// Library/Structures/Cartesian/RobotCartesianPosition
{attribute 'pack_mode' := '1'} 
// ------------------------------------------------------------------------- 
//  SRCI Robot Library                                                
// ------------------------------------------------------------------------- 
//                                                                           
//  Object:      RobotCartesianPosition                                       
//  Author:      Thorsten Brach                                                
//  Date:        2024-06-01
//
//  Description:                                              
//   
//                                                                           
//  Copyright: 
//    (C) 2024 Thorsten Brach. All rights reserved                                                                                                                                            
//             Licensed under the LGPL-3.0 license.
//                                                                           
//  Disclaimer:                                                                           
//    This project is provided without any guarantee and can be used for   
//    private and commercial purposes. Any use is at the user’s 
//    own risk and responsibility.
//
// -------------------------------------------------------------------------
TYPE RobotCartesianPosition EXTENDS RobotCartesianPositionShort : 
STRUCT
  /// Position of second external axis
  E2         : REAL;
  /// Position of third external axis
  E3         : REAL;
  /// Position of fourth external axis
  E4         : REAL;
  /// Position of fifth external axis
  E5         : REAL;
  /// Position of sixth external axis
  E6         : REAL;    
END_STRUCT
END_TYPE

// Library/Structures/Cartesian/RobotCartesianPositionBase
{attribute 'pack_mode' := '1'} 
// ------------------------------------------------------------------------- 
//  SRCI Robot Library                                                
// ------------------------------------------------------------------------- 
//                                                                           
//  Object:      RobotCartesianPosition                                       
//  Author:      Thorsten Brach                                                
//  Date:        2024-06-01
//
//  Description:                                              
//   
//                                                                           
//  Copyright: 
//    (C) 2024 Thorsten Brach. All rights reserved                                                                                                                                            
//             Licensed under the LGPL-3.0 license.
//                                                                           
//  Disclaimer:                                                                           
//    This project is provided without any guarantee and can be used for   
//    private and commercial purposes. Any use is at the user’s 
//    own risk and responsibility.
//
// -------------------------------------------------------------------------
TYPE RobotCartesianPositionBase :
STRUCT
  /// TCP Position on the X-Axis
  X          : REAL;
  /// TCP Position on the Y-Axis
  Y          : REAL;
  /// TCP Position on the Z-Axis
  Z          : REAL;
  /// Rotation around the X-Axis (RX)
  Rx         : REAL;
  /// Rotation around the Y-Axis (RY)
  Ry         : REAL;
  /// Rotation around the Z-Axis (RZ)
  Rz         : REAL;
END_STRUCT
END_TYPE

// Library/Structures/Cartesian/RobotCartesianPositionExt
{attribute 'pack_mode' := '1'} 
// ------------------------------------------------------------------------- 
//  SRCI Robot Library                                                
// ------------------------------------------------------------------------- 
//                                                                           
//  Object:      RobotCartesianPositionExt                                       
//  Author:      Thorsten Brach                                                
//  Date:        2024-06-01
//
//  Description:                                              
//   
//                                                                           
//  Copyright: 
//    (C) 2024 Thorsten Brach. All rights reserved                                                                                                                                            
//             Licensed under the LGPL-3.0 license.
//                                                                           
//  Disclaimer:                                                                           
//    This project is provided without any guarantee and can be used for   
//    private and commercial purposes. Any use is at the user’s 
//    own risk and responsibility.
//
// -------------------------------------------------------------------------
TYPE RobotCartesianPositionExt :
STRUCT
  /// Position of second external axis
  E2 : REAL;
  /// Position of third external axis
  E3 : REAL;
  /// Position of fourth external axis
  E4 : REAL;
  /// Position of fifth external axis
  E5 : REAL;
  /// Position of sixth external axis
  E6 : REAL;  
END_STRUCT
END_TYPE

// Library/Structures/Cartesian/RobotCartesianPositionShort
{attribute 'pack_mode' := '1'} 
// ------------------------------------------------------------------------- 
//  SRCI Robot Library                                                
// ------------------------------------------------------------------------- 
//                                                                           
//  Object:      RobotCartesianPositionShort                                       
//  Author:      Thorsten Brach                                                
//  Date:        2024-06-01
//
//  Description:                                              
//   
//                                                                           
//  Copyright: 
//    (C) 2024 Thorsten Brach. All rights reserved                                                                                                                                            
//             Licensed under the LGPL-3.0 license.
//                                                                           
//  Disclaimer:                                                                           
//    This project is provided without any guarantee and can be used for   
//    private and commercial purposes. Any use is at the user’s 
//    own risk and responsibility.
//
// -------------------------------------------------------------------------
TYPE RobotCartesianPositionShort EXTENDS RobotCartesianPositionBase:
STRUCT
  /// Configuration data of the robot (Config)
  Config     : ArmConfigParameter;
  /// Turn number of the axes (TurnNumber)
  TurnNumber : TurnNumber;
  /// Position of first external axis
  E1         : REAL;
END_STRUCT
END_TYPE

// Library/Structures/Common/CmdHeader
{attribute 'pack_mode' := '1'}
// ------------------------------------------------------------------------- 
//  SRCI Robot Library                                                
// ------------------------------------------------------------------------- 
//                                                                           
//  Object:      CmdHeader                                       
//  Author:      Thorsten Brach                                                
//  Date:        2024-06-01
//
//  Description:                                              
//   
//                                                                           
//  Copyright: 
//    (C) 2024 Thorsten Brach. All rights reserved                                                                                                                                            
//             Licensed under the LGPL-3.0 license.
//                                                                           
//  Disclaimer:                                                                           
//    This project is provided without any guarantee and can be used for   
//    private and commercial purposes. Any use is at the user’s 
//    own risk and responsibility.
//
// ------------------------------------------------------------------------- 
TYPE CmdHeader :
STRUCT
  /// Type of command - For more information see chapter 5.6.4.
 CmdTyp          : CmdType;
 /// Specifies target buffer and processing behavior - For more information see chapter 5.6.4.5
 ExecMode        : ExecutionMode;
 /// Parameter Sequence, used to identify sets of CMD parameter
 ParSeq          : BYTE;
 /// Priority of this command
 Priority        : PriorityLevel;  
END_STRUCT
END_TYPE

// Library/Structures/Common/LogParameter
{attribute 'pack_mode' := '1'} 
// ------------------------------------------------------------------------- 
//  SRCI Robot Library                                                
// ------------------------------------------------------------------------- 
//                                                                           
//  Object:      LogParameter                                       
//  Author:      Thorsten Brach                                                
//  Date:        2024-06-01
//
//  Description:                                              
//   
//                                                                           
//  Copyright: 
//    (C) 2024 Thorsten Brach. All rights reserved                                                                                                                                            
//             Licensed under the LGPL-3.0 license.
//                                                                           
//  Disclaimer:                                                                           
//    This project is provided without any guarantee and can be used for   
//    private and commercial purposes. Any use is at the user’s 
//    own risk and responsibility.
//
// -------------------------------------------------------------------------
TYPE LogParameter :
STRUCT
  /// Log level setting for creating commands  
  CreateCmd : LogLevel;
  /// Log level setting for updating commands
  UpdateCmd : LogLevel;
  /// Log level setting for generating sequence 
  GenSeq    : LogLevel;
  /// Log level for ??? sequence
  DecSeq    : LogLevel;
END_STRUCT
END_TYPE

// Library/Structures/Common/RobotCoordinateSystemParameters
{attribute 'pack_mode' := '1'} 
// ------------------------------------------------------------------------- 
//  SRCI Robot Library                                                
// ------------------------------------------------------------------------- 
//                                                                           
//  Object:      RobotCoordinateSystemParameters                                       
//  Author:      Thorsten Brach                                                
//  Date:        2024-06-01
//
//  Description:                                              
//   
//                                                                           
//  Copyright: 
//    (C) 2024 Thorsten Brach. All rights reserved                                                                                                                                            
//             Licensed under the LGPL-3.0 license.
//                                                                           
//  Disclaimer:                                                                           
//    This project is provided without any guarantee and can be used for   
//    private and commercial purposes. Any use is at the user’s 
//    own risk and responsibility.
//
// -------------------------------------------------------------------------
TYPE RobotCoordinateSystemParameters :
STRUCT
  /// Index of target tool
  /// • 0: Flange (default)
  /// • 1..254: Tool frames
  ToolNo : USINT;
  /// Index of target frame
  /// • 0: WCS (default)
  /// • 1..254: User frames
  FrameNo : USINT;  
END_STRUCT
END_TYPE

// Library/Structures/Common/RspHeader
{attribute 'pack_mode' := '1'}
// ------------------------------------------------------------------------- 
//  SRCI Robot Library                                                
// ------------------------------------------------------------------------- 
//                                                                           
//  Object:      RspHeader                                       
//  Author:      Thorsten Brach                                                
//  Date:        2024-06-01
//
//  Description:                                              
//   
//                                                                           
//  Copyright: 
//    (C) 2024 Thorsten Brach. All rights reserved                                                                                                                                            
//             Licensed under the LGPL-3.0 license.
//                                                                           
//  Disclaimer:                                                                           
//    This project is provided without any guarantee and can be used for   
//    private and commercial purposes. Any use is at the user’s 
//    own risk and responsibility.
//
// -------------------------------------------------------------------------
TYPE RspHeader :  
STRUCT
  /// Parameter Sequence, used to identify sets of CMD parameter - For more information see chapter 5.6.4
  ParSeq               : USINT;
  /// Actual state of the command - For more information and examples, see chapter 5.6.3.2
  State                : CmdMessageState;
  /// Severity of returned message according to .Table 5-47.
  AlarmMessageSeverity : Severity;
  /// Message code for error/warning/info identification reported during execution of command according to
  /// • Error: Table 7-1
  /// • Warning: Table 7-3
  /// • Info: Table 7-5
  AlarmMessageCode     : UINT;  
END_STRUCT
END_TYPE

// Library/Structures/Common/TimeStamp
{attribute 'pack_mode' := '1'} 
// ------------------------------------------------------------------------- 
//  SRCI Robot Library                                                
// ------------------------------------------------------------------------- 
//                                                                           
//  Object:      TimeStamp                                       
//  Author:      Thorsten Brach                                                
//  Date:        2024-06-01
//
//  Description:                                              
//   
//                                                                           
//  Copyright: 
//    (C) 2024 Thorsten Brach. All rights reserved                                                                                                                                            
//             Licensed under the LGPL-3.0 license.
//                                                                           
//  Disclaimer:                                                                           
//    This project is provided without any guarantee and can be used for   
//    private and commercial purposes. Any use is at the user’s 
//    own risk and responsibility.
//
// -------------------------------------------------------------------------
TYPE TimeStamp :
STRUCT
  /// Date of the timestamp
  TsData : IEC_DATE;
  /// Time of the timestamp
  TsTime : IEC_TIME;
END_STRUCT
END_TYPE

// Library/Structures/Data/CyclicStateData
{attribute 'pack_mode' := '1'} 
// ------------------------------------------------------------------------- 
//  SRCI Robot Library                                                
// ------------------------------------------------------------------------- 
//                                                                           
//  Object:      CyclicStateData                                       
//  Author:      Thorsten Brach                                                
//  Date:        2024-06-01
//
//  Description:                                              
//   
//                                                                           
//  Copyright: 
//    (C) 2024 Thorsten Brach. All rights reserved                                                                                                                                            
//             Licensed under the LGPL-3.0 license.
//                                                                           
//  Disclaimer:                                                                           
//    This project is provided without any guarantee and can be used for   
//    private and commercial purposes. Any use is at the user’s 
//    own risk and responsibility.
//
// -------------------------------------------------------------------------
TYPE CyclicStateData :
STRUCT
  /// Combination of various RA related states.
  StatusWord : RaStatusWord;
  /// Actual override in percentage multiplied by 100 (see chapter 5.6.2 for more information about the percentage encoding)
  Override   : UINT;
END_STRUCT
END_TYPE

// Library/Structures/Data/FrameData
{attribute 'pack_mode' := '1'} 
// ------------------------------------------------------------------------- 
//  SRCI Robot Library                                                
// ------------------------------------------------------------------------- 
//                                                                           
//  Object:      FrameData                                       
//  Author:      Thorsten Brach                                                
//  Date:        2024-06-01
//
//  Description:                                              
//   
//                                                                           
//  Copyright: 
//    (C) 2024 Thorsten Brach. All rights reserved                                                                                                                                            
//             Licensed under the LGPL-3.0 license.
//                                                                           
//  Disclaimer:                                                                           
//    This project is provided without any guarantee and can be used for   
//    private and commercial purposes. Any use is at the user’s 
//    own risk and responsibility.
//
// -------------------------------------------------------------------------
TYPE FrameData :
STRUCT
  /// Timestamp
  Timestamp      : IEC_TIMESTAMP;
  /// Frame to which the shifting and rotation is relative M
  ReferenceFrame : USINT;
  /// Origin of the coordinate system relative to the BCS/WCS/UCS 
  /// X value [mm]  
  X              : REAL := 0;
  /// Origin of the coordinate system relative to the BCS/WCS/UCS 
  /// Y value [mm]  
  Y              : REAL := 0;
  /// Origin of the coordinate system relative to the BCS/WCS/UCS 
  /// Z value [mm]  
  Z              : REAL := 0;
  /// Orientation of the coordinate system relative to the BCS/WCS/UCS
  /// Rx value [°]  
  Rx             : REAL := 0;
  /// Rx value [°]  
  Ry             : REAL := 0;
  /// Rx value [°]  
  Rz             : REAL := 0;  
END_STRUCT
END_TYPE

// Library/Structures/Data/LoadData
{attribute 'pack_mode' := '1'} 
// ------------------------------------------------------------------------- 
//  SRCI Robot Library                                                
// ------------------------------------------------------------------------- 
//                                                                           
//  Object:      LoadData                                       
//  Author:      Thorsten Brach                                                
//  Date:        2024-06-01
//
//  Description:                                              
//   
//                                                                           
//  Copyright: 
//    (C) 2024 Thorsten Brach. All rights reserved                                                                                                                                            
//             Licensed under the LGPL-3.0 license.
//                                                                           
//  Disclaimer:                                                                           
//    This project is provided without any guarantee and can be used for   
//    private and commercial purposes. Any use is at the user’s 
//    own risk and responsibility.
//
// -------------------------------------------------------------------------
TYPE LoadData :
STRUCT
  /// Timestamp
  Timestamp : IEC_TIMESTAMP;
  /// Position of the center of gravity relative to the flange.
  /// X value [mm]  
  X         : REAL := 0;
  /// Position of the center of gravity relative to the flange.
  /// Y value [mm]  
  Y         : REAL := 0;
  /// Position of the center of gravity relative to the flange.
  /// Z value [mm]  
  Z         : REAL := 0;
  /// Orientation of the principal inertia axes relative to the flange. O
  /// Rx value [°]  
  Rx        : REAL := 0;
  /// Ry value [°]  
  Ry        : REAL := 0;
  /// Rz value [°]  
  Rz        : REAL := 0;
  /// The mass of the tool and workpiece being gripped. [kg]
  Mass      : REAL := 0;
  /// The moment of inertia of the load around the resulting inertia X-Axis [kg/m²]
  Ix        : REAL := 0;
  /// The moment of inertia of the load around the resulting inertia y-axis [kg/m²]
  Iy        : REAL := 0;
  /// The moment of inertia of the load around the resulting inertia z-axis [kg/m²]
  Iz        : REAL := 0;  
END_STRUCT
END_TYPE

// Library/Structures/Data/RobotSubProgramData
{attribute 'pack_mode' := '1'} 
// ------------------------------------------------------------------------- 
//  SRCI Robot Library                                                
// ------------------------------------------------------------------------- 
//                                                                           
//  Object:      RobotSubProgramData                                       
//  Author:      Thorsten Brach                                                
//  Date:        2024-06-01
//
//  Description:                                              
//   
//                                                                           
//  Copyright: 
//    (C) 2024 Thorsten Brach. All rights reserved                                                                                                                                            
//             Licensed under the LGPL-3.0 license.
//                                                                           
//  Disclaimer:                                                                           
//    This project is provided without any guarantee and can be used for   
//    private and commercial purposes. Any use is at the user’s 
//    own risk and responsibility.
//
// -------------------------------------------------------------------------
TYPE RobotSubProgramData :
STRUCT
  /// Sub program data
  Data : ARRAY [0..25] OF BYTE;
END_STRUCT
END_TYPE

// Library/Structures/Data/SplineData
{attribute 'pack_mode' := '1'} 
// ------------------------------------------------------------------------- 
//  SRCI Robot Library                                                
// ------------------------------------------------------------------------- 
//                                                                           
//  Object:      SplineData                                       
//  Author:      Thorsten Brach                                                
//  Date:        2024-06-01
//
//  Description:                                              
//   
//                                                                           
//  Copyright: 
//    (C) 2024 Thorsten Brach. All rights reserved                                                                                                                                            
//             Licensed under the LGPL-3.0 license.
//                                                                           
//  Disclaimer:                                                                           
//    This project is provided without any guarantee and can be used for   
//    private and commercial purposes. Any use is at the user’s 
//    own risk and responsibility.
//
// -------------------------------------------------------------------------
TYPE SplineData :
STRUCT
    /// Absolute target coordinates in the selected coordinate system (see ToolNo and FrameNo).
    Position         : RobotCartesianPosition;
    /// TCP velocity in % of nominal velocity.
    /// •  <0% : Use default velocity (default)
    /// •   0% : Use internal minimal velocity
    /// • 100% : Use maximal reference velocity
    /// • See chapter 5.5.7 Robot dynamics
    VelocityRate     : REAL;    
    /// Acceleration for movement in % of nominal acceleration.
    /// •  <0% : Use default acceleration (default)
    /// •   0% : Use internal minimal acceleration
    /// • 100% : Use maximal reference acceleration
    /// • See chapter 5.5.7 Robot dynamics
    AccelerationRate : REAL;    
    /// Deceleration for movement in % of nominal deceleration.
    /// •  <0% : Use default deceleration (default)
    /// •   0% : Use internal minimal deceleration
    /// • 100% : Use maximal reference deceleration
    /// • See chapter 5.5.7 Robot dynamics
    DecelerationRate : REAL;    
    /// Jerk of the movement in % of nominal jerk.
    /// <0% o Use default jerk (default)
    /// 0% o Use internal minimal jerk
    /// 100% o Use maximal reference jerk
    /// See chapter 5.5.7 Robot dynamics
    JerkRate         : REAL;
    /// Index of tool
    /// 0: Flange (default)
    /// 1..254: Tool frames
    ToolNo           : USINT;    
    /// Index of frame
    /// 0: WCS (default)
    /// 1..254: User frames
    FrameNo          : USINT;    
    /// [ms] Parameter is used if it is greater than 0 (default):
    /// Parameter defines the time for the movement to reach the target position
    /// Velocity input can be ignored
    /// Acceleration, Deceleration and jerk will be ignored
    /// Define two consecutive points with identical positions and specified Time to realize waiting time on spline.
    /// Error is sent by the RC, if the time cannot be kept.
    MoveTime         : TIME;  
END_STRUCT
END_TYPE

// Library/Structures/Data/ToolData
{attribute 'pack_mode' := '1'} 
// ------------------------------------------------------------------------- 
//  SRCI Robot Library                                                
// ------------------------------------------------------------------------- 
//                                                                           
//  Object:      ToolData                                       
//  Author:      Thorsten Brach                                                
//  Date:        2024-06-01
//
//  Description:                                              
//   
//                                                                           
//  Copyright: 
//    (C) 2024 Thorsten Brach. All rights reserved                                                                                                                                            
//             Licensed under the LGPL-3.0 license.
//                                                                           
//  Disclaimer:                                                                           
//    This project is provided without any guarantee and can be used for   
//    private and commercial purposes. Any use is at the user’s 
//    own risk and responsibility.
//
// -------------------------------------------------------------------------
TYPE ToolData :
STRUCT
  /// Timestamp
  Timestamp   : IEC_TIMESTAMP;
  /// Identification of physical tool Default: 0 
  ID          : USINT;
  /// True: Tool fixed False: Tool on flange 
  ExternalTCP : BOOL;
  /// Origin of the tool coordinate system relative to the flange coordinate system. 
  /// X value [mm]  
  X           : REAL;
  /// Origin of the tool coordinate system relative to the flange coordinate system. 
  /// Y value [mm]  
  Y           : REAL;
  /// Origin of the tool coordinate system relative to the flange coordinate system. 
  /// Z value [mm]  
  Z           : REAL;
  /// Orientation of the tool coordinate system relative to the flange coordinate system 
  /// RX value[°]
  Rx          : REAL;
  /// Orientation of the tool coordinate system relative to the flange coordinate system 
  /// RX value[°]
  Ry          : REAL;
  /// Orientation of the tool coordinate system relative to the flange coordinate system 
  /// RX value[°]
  Rz          : REAL;
  /// Index of the payload Information of tool and workpiece weight, center of gravity and inertia 
  LoadNo      : USINT;  
END_STRUCT
END_TYPE

// Library/Structures/Data/UserData
{attribute 'pack_mode' := '1'} 
// ------------------------------------------------------------------------- 
//  SRCI Robot Library                                                
// ------------------------------------------------------------------------- 
//                                                                           
//  Object:      UserData                                       
//  Author:      Thorsten Brach                                                
//  Date:        2024-06-01
//
//  Description:                                              
//   
//                                                                           
//  Copyright: 
//    (C) 2024 Thorsten Brach. All rights reserved                                                                                                                                            
//             Licensed under the LGPL-3.0 license.
//                                                                           
//  Disclaimer:                                                                           
//    This project is provided without any guarantee and can be used for   
//    private and commercial purposes. Any use is at the user’s 
//    own risk and responsibility.
//
// -------------------------------------------------------------------------
TYPE UserData :
STRUCT
  /// Set TRUE (default), to activate the synchronizationrelated comparison mechanism for tool data 
  EnableSyncTool                 : BOOL;
  /// Set TRUE (default), to activate the synchronizationrelated comparison mechanism for frame data
  EnableSyncFrame                : BOOL;
  /// Set TRUE (default), to activate the synchronizationrelated comparison mechanism for load data
  EnableSyncLoad                 : BOOL;
  /// Set TRUE (default), to activate the synchronizationrelated comparison mechanism for work area data
  EnableSyncWorkArea             : BOOL;
  /// Set TRUE (default), to activate the synchronizationrelated comparison mechanism for software limits
  EnableSyncSWLimits             : BOOL;
  /// Set TRUE (default), to activate the synchronizationrelated comparison mechanism for default dynamics
  EnableSyncDefaultDynamics      : BOOL;
  /// Set TRUE (default), to activate the synchronizationrelated comparison mechanism for reference dynamics
  EnableSyncReferenceDynamics    : BOOL;
  /// Set TRUE to define two sequences in one Telegram.
  ActivateTwoSequences           : BOOL;
  /// Define direction of synchronization for tool data according to Table 6-4
  SyncModeTool                   : SINT;
  /// Define direction of synchronization for frame data according to Table 6-4  
  SyncModeFrame                  : SINT;
  /// Define direction of synchronization for load data according to Table 6-4
  SyncModeLoad                   : SINT;
  /// Define direction of synchronization for work area data according to Table 6-4
  SyncModeWorkAreas              : SINT;
  /// Define direction of synchronization for software limits according to Table 6-4
  SyncModeSWLimits               : SINT;
  /// Define direction of synchronization for default dynamics according to Table 6-4
  SyncModeDefaultDynamics        : SINT;
  /// Define direction of synchronization for reference dynamics according to Table 6-4
  SyncModeReferenceDynamics      : SINT;
  /// Defines waiting time [ms] of RC between receiving a first move command when motion queue is empty and starting the first movement. See also chapter 5.6.8.
  DelayTime                      : UINT; 
  /// Define number of points required to calculate the blending. See also chapter 5.6.8
  WaitForNrOfCmd                 : UINT;
  ///Defines blending behavior for single move commands
  /// • 0 (default): Move to end position :
  ///     Robot moves exactly the target position independently of the selected "BlendingMode"
  /// 
  /// • 1: Wait at blending parameter : 
  ///      Robot stops its movement when the specified blending parameter is reached
  WaitAtBlendingZone             : BOOL;
  /// Allow a sequence switch from primary to secondary while a subprogram called via CallSubprogram (6.5.18) in the sequence is in progress
  AllowSecSeqWhileSubprogram     : BOOL;
  /// Allows blending when CallSubprogram is called in sequence and removed afterwards.
  /// For more information see chapter 6.5.21.
  /// • 0 (default): Dynamic blending is prevented
  /// • 1: Dynamic blending is allowed
  AllowDynamicBlending           : BOOL;
  /// Maximum allowed time [ms] between incrementation of LifeSign before communication error.
  /// • <10 ms: Invalid
  /// • 50 ms: default
  /// See also chapter 5.6.6.2.
  LifeSignTimeOut                : UINT;
  /// Specifies system reaction in case inconsistency of synchronization data is detected according to Table 6-81. For more information refer to chapter 5.6.7.2
  SyncReaction                   : USINT;
  /// Defines a delay time [ms] between detecting an inconsistency of configuration data between server and client an executing the defined SyncReaction.
  /// Always positive.
  /// • Default: 0 ms
  SyncDelay                      : UINT;
  /// Defines up to which level of severity messages will be logged in the RC's server log
  LogLevel                       : LogLevel;
  /// Defines up to which level of severity messages will be transmitted to the PLC’s message buffer
  MessageLevel                   : MessageLevel;
  /// Version of client implementation in format (X.X.X)
  PLCLibraryVersion              : VersionStruct;
  /// RC manufacturer name 
  RCManufacturer                 : STRING(20); 
  /// RC part number 
  RCOrderID                      : STRING(20); 
  /// RC serial number 
  RCSerialNumber                 : STRING(16); 
  /// RA serial number 
  RASerialNumber                 : STRING(16); 
  /// Robot firmware version in manufacturer-specific format 
  RCFirmwareVersion              : STRING(12); 
  /// Version of server implementation in format (X.X.X) 
  RCInterpreterVersion           : VersionStruct;
  /// Version of SRCI specification on which server implementation is based in format (X.X.X)  
  RCSRCIVersion                  : VersionStruct;
  /// TRUE  = Axis used in Robot, FALSE = Axis NOT used. See Table 6-13 for bit assignment.
  AxisJointUsed                  : BYTE;
  /// TRUE = Axis used by Robot, FALSE = Axis NOT used. See Table 6-13 for bit assignment.
  AxisExternalUsed               : BYTE;
  /// TRUE = mm, FALSE = °. See Table 6-13 for bit assignment.
  AxisJointUnit                  : BYTE;
  /// TRUE = mm, FALSE = °. See Table 6-13 for bit assignment.
  AxisExternalUnit               : BYTE;
  /// Interface is initialized and ready to process commands.
  Initialized                    : BOOL;
  /// All synchronization-related configuration data between client and server is synchronized.
  Synchronized                   : BOOL;
  /// ToolData synchronization is activated.
  ToolDataSynchronizing          : BOOL;
  /// FrameData synchronization is activated.
  FrameDataSynchronizing         : BOOL;
  /// LoadData synchronization is activated.
  LoadDataSynchronizing          : BOOL;
  /// WorkAreaData synchronization is activated.
  WorkAreaDataSynchronizing      : BOOL;
  /// SWLimits synchronization is activated.
  SWLimitsSynchronizing          : BOOL;
  /// DefaultDynamics synchronization is activated.
  DefaultDynamicsSynchronizing   : BOOL;
  /// ReferenceDynamics synchronization is activated.
  ReferenceDynamicsSynchronizing : BOOL;
  /// TRUE, when robot’s axes values change due to physical movement of axes. Can only be TRUE in sequence state "Executing". Default: FALSE 
  IsMoving                       : BOOL;
  /// TRUE, when move commands buffered by the primary sequence are currently not processed. Default: FALSE 
  PrimarySequencePaused          : BOOL;
  /// TRUE, when robot is moving in the primary sequence. FALSE, when robot leaves its position by other means than move commands in the primary sequence. Default: FALSE
  InPrimaryPos                   : BOOL;
  /// TRUE, when secondary sequence is active. Default: FALSE
  SecondarySequenceActive        : BOOL;
  /// Shows that an error acknowledgement by the client is necessary. Default: FALSE
  ErrorPending                   : BOOL;
  /// TRUE, when RC is restarting. Default: FALSE
  RestartInProgress              : BOOL;
  /// Signals that a brake test is required in the defined monitoring time (see chapter 6.5.27).
  BrakeTestRequired              : BOOL;
  /// RA power state. Default: FALSE
  Enabled                        : BOOL;
  /// TRUE, while RA sequence states returns Idle. Default: FALSE
  Idle                           : BOOL;
  /// TRUE, while RA sequence states returns Executing. Default: FALSE
  Executing                      : BOOL;
  /// TRUE, while RA sequence states returns Interrupted. Default: FALSE
  Interrupted                    : BOOL;
  /// TRUE, when robot is currently blending between to move commands. Can only be TRUE in sequence state "Executing". Default: FALSE
  IsBlending                     : BOOL;  
  /// Operation Mode (see chapter 5.5.1)
  OperationMode                  : USINT;
  /// PathAccuracyMode is active (see chapter 6.5.22) 
  PathAccuracyMode               : BOOL;
  /// AvoidSingularity is active (see chapter 6.5.23) 
  AvoidSingularity               : BOOL;
  /// TRUE, while CollisionDetection is enabled (see chapter 6.5.35) Default: FALSE 
  CollisionDetectionEnabled      : BOOL;
  /// TRUE, when a collision was detected while CollisionDetection is enabled (see chapter 6.5.35) Default: FALSE 
  CollisionDetected              : BOOL;
  /// TRUE, when the RC requests a restart of the RC induced through the functions "WriteRobotSWLimits" (chapter 6.2.16) or "WriteSystemVariable" (chapter 6.5.8) Default: FALSE 
  RestartRequested               : BOOL;
  /// Actual override
  ActualOverride                 : UINT;
  /// StepMode is active and set to ExactStop (see chapter 6.1.3) 
  StepModeExactStopActive        : BOOL;
  /// StepMode is active and set to Blending (see chapter 6.1.3) 
  StepModeBlendingActive         : BOOL;
  /// Cyclic dynamics status bit Accelerating is supported by RC (see chapter 5.5.3.2) 
  AcceleratingSupported          : BOOL;
  /// TRUE, when the robot is currently accelerating Default: FALSE 
  Accelerating                   : BOOL;
  /// Cyclic dynamics status bit Decelerating is supported by RC (see chapter 5.5.3.2) 
  DeceleratingSupported          : BOOL;
  /// TRUE, when the robot is currently decelerating Default: FALSE 
  Decelerating                   : BOOL;
  /// Cyclic dynamics status bit ConstantVelocity is supported by RC (see chapter 5.5.3.2) 
  ConstantVelocitySupported      : BOOL;
  /// TRUE, while the robot velocity is constant Default: FALSE 
  ConstantVelocity               : BOOL;
  /// TRUE, while the CartesianPosition is returned cyclically 
  ReadingCartesianPosition       : BOOL;
  /// TRUE, while the ExtCartesianPosition is returned cyclically 
  ReadingExtCartesianPosition    : BOOL;
  /// TRUE, while the JointPosition is returned cyclically 
  ReadingJointPosition           : BOOL;
  /// TRUE, while the ExtJointPosition is returned cyclically 
  ReadingExtJointPosition        : BOOL;
  /// Cyclically returned, absolute coordinates of current position in selected coordinate systems (see input parameters ToolNo and FrameNo of function ReadActualPositionCyclic 6.1.6)
  CartesianPosition              : RobotCartesianPositionShort;
  /// Cyclically returned, absolute cartesian position of the external axes of the robot in selected coordinate systems (see input parameters ToolNo and FrameNo of function ReadActualPositionCyclic 6.1.6)
  ExtCartesianPosition           : RobotCartesianPositionExt;  
  /// Cyclically returned, absolute position of the robot in Joint position
  JointPosition                  : RobotJointPositionShort;
  /// Cyclically returned, absolute joint position of the external axes of the robot
  ExtJointPosition               : RobotJointPositionExt;
  /// TRUE: Function is supported by RC
  /// FALSE: Function is not supported by RC
  /// See Table 6-14 for bit assignment.
  RCSupportedFunctions           : RCSupportedFunctions;
END_STRUCT
END_TYPE

// Library/Structures/DatenAndTime/IEC_DATE
/// Date in the format days since 1990.01.01
TYPE IEC_DATE : UINT; 
// ------------------------------------------------------------------------- 
//  SRCI Robot Library                                                
// ------------------------------------------------------------------------- 
//                                                                           
//  Object:      IEC_DATE                                       
//  Author:      Thorsten Brach                                                
//  Date:        2024-06-01
//
//  Description:                                              
//   
//                                                                           
//  Copyright: 
//    (C) 2024 Thorsten Brach. All rights reserved                                                                                                                                            
//             Licensed under the LGPL-3.0 license.
//                                                                           
//  Disclaimer:                                                                           
//    This project is provided without any guarantee and can be used for   
//    private and commercial purposes. Any use is at the user’s 
//    own risk and responsibility.
//
// -------------------------------------------------------------------------
END_TYPE

// Library/Structures/DatenAndTime/IEC_TIME
/// Time in the clients time zone in the format milliseconds since start of day
TYPE IEC_TIME : TIME_OF_DAY; 
// ------------------------------------------------------------------------- 
//  SRCI Robot Library                                                
// ------------------------------------------------------------------------- 
//                                                                           
//  Object:      IEC_TIME                                       
//  Author:      Thorsten Brach                                                
//  Date:        2024-06-01
//
//  Description:                                              
//   
//                                                                           
//  Copyright: 
//    (C) 2024 Thorsten Brach. All rights reserved                                                                                                                                            
//             Licensed under the LGPL-3.0 license.
//                                                                           
//  Disclaimer:                                                                           
//    This project is provided without any guarantee and can be used for   
//    private and commercial purposes. Any use is at the user’s 
//    own risk and responsibility.
//
// -------------------------------------------------------------------------
END_TYPE

// Library/Structures/DatenAndTime/IEC_TIMESTAMP
TYPE IEC_TIMESTAMP :
// ------------------------------------------------------------------------- 
//  SRCI Robot Library                                                
// ------------------------------------------------------------------------- 
//                                                                           
//  Object:      IEC_TimeStamp                                       
//  Author:      Thorsten Brach                                                
//  Date:        2024-06-11
//
//  Description:                                              
//   
//                                                                           
//  Copyright: 
//    (C) 2024 Thorsten Brach. All rights reserved                                                                                                                                            
//             Licensed under the LGPL-3.0 license.
//                                                                           
//  Disclaimer:                                                                           
//    This project is provided without any guarantee and can be used for   
//    private and commercial purposes. Any use is at the user’s 
//    own risk and responsibility.
//
// -------------------------------------------------------------------------
STRUCT
  /// Date
  IEC_DATE : IEC_DATE;
  /// Time
  IEC_TIME : IEC_TIME;
END_STRUCT
END_TYPE

// Library/Structures/DatenAndTime/SystemTime
TYPE SystemTime :
// ------------------------------------------------------------------------- 
//  SRCI Robot Library                                                
// ------------------------------------------------------------------------- 
//                                                                           
//  Object:      SystemTime                                       
//  Author:      Thorsten Brach                                                
//  Date:        2025-01-11
//
//  Description:                                              
//   
//                                                                           
//  Copyright: 
//    (C) 2025 Thorsten Brach. All rights reserved                                                                                                                                            
//             Licensed under the LGPL-3.0 license.
//                                                                           
//  Disclaimer:                                                                           
//    This project is provided without any guarantee and can be used for   
//    private and commercial purposes. Any use is at the user’s 
//    own risk and responsibility.
//
// -------------------------------------------------------------------------  
STRUCT
  /// Date of the system
  SystemDate : DATE;
  /// Time of the system
  SystemTime : TOD; 
END_STRUCT
END_TYPE

// Library/Structures/Dynamics/DefaultDynamics
{attribute 'pack_mode' := '1'} 
// ------------------------------------------------------------------------- 
//  SRCI Robot Library                                                
// ------------------------------------------------------------------------- 
//                                                                           
//  Object:      DefaultDynamics                                       
//  Author:      Thorsten Brach                                                
//  Date:        2024-06-01
//
//  Description:                                              
//   
//                                                                           
//  Copyright: 
//    (C) 2024 Thorsten Brach. All rights reserved                                                                                                                                            
//             Licensed under the LGPL-3.0 license.
//                                                                           
//  Disclaimer:                                                                           
//    This project is provided without any guarantee and can be used for   
//    private and commercial purposes. Any use is at the user’s 
//    own risk and responsibility.
//
// -------------------------------------------------------------------------
TYPE DefaultDynamics :
STRUCT
  /// Timestamp
  Timestamp        : IEC_TIMESTAMP;
  /// Maximum velocity for the axes.
  /// Range [%]: 
  /// •  <0% : Use default velocity given by the user
  /// •   0% : Use internal minimal velocity
  /// • 100% : Use the entire reference velocity, given by the user
  VelocityRate     : REAL;
  /// Maximum acceleration.
  /// Range [%]:
  /// •  <0% : Use default acceleration given by the user
  /// •   0% : Use internal minimal acceleration
  /// • 100% : Use the entire reference acceleration, given by the user
  AccelerationRate : REAL;
  /// Maximum deceleration.
  /// Range [%] : 
  /// •  <0% : Use default deceleration given by the user
  /// •   0% : Use internal minimal deceleration
  /// • 100% : Use the entire reference deceleration, given by the user
  DecelerationRate : REAL;
  /// Maximum jerk
  /// Range [%] : 
  /// •  <0% : Use default jerk given by the user
  /// •   0% : Use internal minimal jerk
  /// • 100% : Use the entire reference jerk, given by the user (Trapezoidal if possible) 
  JerkRate         : REAL;  
END_STRUCT
END_TYPE

// Library/Structures/Dynamics/ReferenceDynamics
{attribute 'pack_mode' := '1'}
// ------------------------------------------------------------------------- 
//  SRCI Robot Library                                                
// ------------------------------------------------------------------------- 
//                                                                           
//  Object:      ReferenceDynamics                                       
//  Author:      Thorsten Brach                                                
//  Date:        2024-06-01
//
//  Description:                                              
//   
//                                                                           
//  Copyright: 
//    (C) 2024 Thorsten Brach. All rights reserved                                                                                                                                            
//             Licensed under the LGPL-3.0 license.
//                                                                           
//  Disclaimer:                                                                           
//    This project is provided without any guarantee and can be used for   
//    private and commercial purposes. Any use is at the user’s 
//    own risk and responsibility.
//
// ------------------------------------------------------------------------- 
TYPE ReferenceDynamics :
STRUCT
  /// Timestamp
  Timestamp             : IEC_TIMESTAMP;
  /// Path velocity [mm/s](tangent) at 100%
  /// • <0: (default) - Do not change values
  /// • ≥0: Change values according to input value
  VelocityReference     : REAL;
  /// Path acceleration [mm/s2] at 100%
  /// • <0: (default) - Do not change values
  /// • ≥0: Change values according to input value
  AccelerationReference : REAL;
  /// Path deceleration [mm/s2] at 100%
  /// • <0: (default) - Do not change values
  /// • ≥0: Change values according to input value
  DecelerationReference : REAL;
  /// Jerk [mm/s3] at 100%
  /// • <0: (default) - Do not change values
  /// • ≥0: Change values according to input value
  JerkReference        : REAL;  
END_STRUCT
END_TYPE

// Library/Structures/Joint/RobotJointCurrent
{attribute 'pack_mode' := '1'} 
// ------------------------------------------------------------------------- 
//  SRCI Robot Library                                                
// ------------------------------------------------------------------------- 
//                                                                           
//  Object:      RobotJointCurrent                                       
//  Author:      Thorsten Brach                                                
//  Date:        2024-06-01
//
//  Description:                                              
//   
//                                                                           
//  Copyright: 
//    (C) 2024 Thorsten Brach. All rights reserved                                                                                                                                            
//             Licensed under the LGPL-3.0 license.
//                                                                           
//  Disclaimer:                                                                           
//    This project is provided without any guarantee and can be used for   
//    private and commercial purposes. Any use is at the user’s 
//    own risk and responsibility.
//
// -------------------------------------------------------------------------
TYPE RobotJointCurrent :
STRUCT
  /// Current of first joint of the robot
  J1 : REAL;
  /// Current of second joint of the robot
  J2 : REAL;
  /// Current of third joint of the robot
  J3 : REAL;
  /// Current of fourth joint of the robot
  J4 : REAL;
  /// Current of fifth joint of the robot
  J5 : REAL;
  /// Current of sixth joint of the robot
  J6 : REAL;
  /// Current of first external joint of the robot
  E1 : REAL;
  /// Current of second external axis
  E2: REAL;
  /// Current of third external axis
  E3: REAL;
  /// Current of fourth external axis
  E4: REAL;
  /// Current of fifth external axis
  E5: REAL;
  /// Current of sixth external axis
  E6: REAL;  
END_STRUCT
END_TYPE

// Library/Structures/Joint/RobotJointCurrentExt
{attribute 'pack_mode' := '1'} 
// ------------------------------------------------------------------------- 
//  SRCI Robot Library                                                
// ------------------------------------------------------------------------- 
//                                                                           
//  Object:      RobotJointCurrentExt                                       
//  Author:      Thorsten Brach                                                
//  Date:        2024-06-01
//
//  Description:                                              
//   
//                                                                           
//  Copyright: 
//    (C) 2024 Thorsten Brach. All rights reserved                                                                                                                                            
//             Licensed under the LGPL-3.0 license.
//                                                                           
//  Disclaimer:                                                                           
//    This project is provided without any guarantee and can be used for   
//    private and commercial purposes. Any use is at the user’s 
//    own risk and responsibility.
//
// -------------------------------------------------------------------------
TYPE RobotJointCurrentExt :
STRUCT
  /// Current of first external joint of the robot
  E1 : REAL;
  /// Current of second external axis
  E2: REAL;
  /// Current of third external axis
  E3: REAL;
  /// Current of fourth external axis
  E4: REAL;
  /// Current of fifth external axis
  E5: REAL;
  /// Current of sixth external axis
  E6: REAL;  
END_STRUCT
END_TYPE

// Library/Structures/Joint/RobotJointCurrentShort
{attribute 'pack_mode' := '1'} 
// ------------------------------------------------------------------------- 
//  SRCI Robot Library                                                
// ------------------------------------------------------------------------- 
//                                                                           
//  Object:      RobotJointCurrentShort                                       
//  Author:      Thorsten Brach                                                
//  Date:        2024-06-01
//
//  Description:                                              
//   
//                                                                           
//  Copyright: 
//    (C) 2024 Thorsten Brach. All rights reserved                                                                                                                                            
//             Licensed under the LGPL-3.0 license.
//                                                                           
//  Disclaimer:                                                                           
//    This project is provided without any guarantee and can be used for   
//    private and commercial purposes. Any use is at the user’s 
//    own risk and responsibility.
//
// -------------------------------------------------------------------------
TYPE RobotJointCurrentShort :
STRUCT
  /// Current of first joint of the robot
  J1 : REAL;
  /// Current of second joint of the robot
  J2 : REAL;
  /// Current of third joint of the robot
  J3 : REAL;
  /// Current of fourth joint of the robot
  J4 : REAL;
  /// Current of fifth joint of the robot
  J5 : REAL;
  /// Current of sixth joint of the robot
  J6 : REAL;
END_STRUCT
END_TYPE

// Library/Structures/Joint/RobotJointPosition
{attribute 'pack_mode' := '1'} 
// ------------------------------------------------------------------------- 
//  SRCI Robot Library                                                
// ------------------------------------------------------------------------- 
//                                                                           
//  Object:      RobotJointPosition                                       
//  Author:      Thorsten Brach                                                
//  Date:        2024-06-01
//
//  Description:                                              
//   
//                                                                           
//  Copyright: 
//    (C) 2024 Thorsten Brach. All rights reserved                                                                                                                                            
//             Licensed under the LGPL-3.0 license.
//                                                                           
//  Disclaimer:                                                                           
//    This project is provided without any guarantee and can be used for   
//    private and commercial purposes. Any use is at the user’s 
//    own risk and responsibility.
//
// -------------------------------------------------------------------------
TYPE RobotJointPosition :
STRUCT
  /// Position [°] of first joint of the robot
  J1 : REAL;
  /// Position [°] of second joint of the robot
  J2 : REAL;
  /// Position [°] of third joint of the robot
  J3 : REAL;
  /// Position [°] of fourth joint of the robot
  J4 : REAL;
  /// Position [°] of fifth joint of the robot
  J5 : REAL;
  /// Position [°] of sixth joint of the robot
  J6 : REAL;
  /// Position [°] of first external axis 
  E1 : REAL;  
  /// Position [°] of second external axis
  E2 : REAL;
  /// Position [°] of third external axis
  E3 : REAL;
  /// Position [°] of fourth external axis
  E4 : REAL;
  /// Position [°] of fifth external axis
  E5 : REAL;
  /// Position [°] of sixth external axis
  E6 : REAL;  
END_STRUCT
END_TYPE

// Library/Structures/Joint/RobotJointPositionExt
{attribute 'pack_mode' := '1'} 
// ------------------------------------------------------------------------- 
//  SRCI Robot Library                                                
// ------------------------------------------------------------------------- 
//                                                                           
//  Object:      RobotJointPositionExt                                       
//  Author:      Thorsten Brach                                                
//  Date:        2024-06-01
//
//  Description:                                              
//   
//                                                                           
//  Copyright: 
//    (C) 2024 Thorsten Brach. All rights reserved                                                                                                                                            
//             Licensed under the LGPL-3.0 license.
//                                                                           
//  Disclaimer:                                                                           
//    This project is provided without any guarantee and can be used for   
//    private and commercial purposes. Any use is at the user’s 
//    own risk and responsibility.
//
// -------------------------------------------------------------------------
TYPE RobotJointPositionExt :
STRUCT
  /// Position of second external axis
  E2: REAL;
  /// Position of third external axis
  E3: REAL;
  /// Position of fourth external axis
  E4: REAL;
  /// Position of fifth external axis
  E5: REAL;
  /// Position of sixth external axis
  E6: REAL;  
END_STRUCT
END_TYPE

// Library/Structures/Joint/RobotJointPositionShort
{attribute 'pack_mode' := '1'} 
// ------------------------------------------------------------------------- 
//  SRCI Robot Library                                                
// ------------------------------------------------------------------------- 
//                                                                           
//  Object:      RobotJointPositionShort                                       
//  Author:      Thorsten Brach                                                
//  Date:        2024-06-01
//
//  Description:                                              
//   
//                                                                           
//  Copyright: 
//    (C) 2024 Thorsten Brach. All rights reserved                                                                                                                                            
//             Licensed under the LGPL-3.0 license.
//                                                                           
//  Disclaimer:                                                                           
//    This project is provided without any guarantee and can be used for   
//    private and commercial purposes. Any use is at the user’s 
//    own risk and responsibility.
//
// -------------------------------------------------------------------------
TYPE RobotJointPositionShort :
STRUCT
  /// Position of first joint of the robot
  J1 : REAL;
  /// Position of second joint of the robot
  J2 : REAL;
  /// Position of third joint of the robot
  J3 : REAL;
  /// Position of fourth joint of the robot
  J4 : REAL;
  /// Position of fifth joint of the robot
  J5 : REAL;
  /// Position of sixth joint of the robot
  J6 : REAL;
  /// Position of first external axis 
  E1 : REAL;  
END_STRUCT
END_TYPE

// Library/Structures/Miscellaneous/AlarmMessage
{attribute 'pack_mode' := '1'} 
// ------------------------------------------------------------------------- 
//  SRCI Robot Library                                                
// ------------------------------------------------------------------------- 
//                                                                           
//  Object:      AlarmMessage                                       
//  Author:      Thorsten Brach                                                
//  Date:        2024-06-01
//
//  Description:                                              
//   
//                                                                           
//  Copyright: 
//    (C) 2024 Thorsten Brach. All rights reserved                                                                                                                                            
//             Licensed under the LGPL-3.0 license.
//                                                                           
//  Disclaimer:                                                                           
//    This project is provided without any guarantee and can be used for   
//    private and commercial purposes. Any use is at the user’s 
//    own risk and responsibility.
//
// -------------------------------------------------------------------------
TYPE AlarmMessage :
STRUCT
  /// Timestamp
  Timestamp   : SystemTime;
  /// Type of message according to Table 5-46:
  MessageType : MessageType;
  /// Severity of message according to Table 5-47: Debug, Info, Warning, Error, Fatal error
  Severity    : Severity;
  /// Code of messages
  MessageCode : DWORD;
  /// Static text of message
  MessageText : STRING(255);  
END_STRUCT
END_TYPE

// Library/Structures/Miscellaneous/ArmConfigParameter
{attribute 'pack_mode' := '1'} 
// ------------------------------------------------------------------------- 
//  SRCI Robot Library                                                
// ------------------------------------------------------------------------- 
//                                                                           
//  Object:      ArmConfigParameter                                       
//  Author:      Thorsten Brach                                                
//  Date:        2024-06-01
//
//  Description:                                              
//   
//                                                                           
//  Copyright: 
//    (C) 2024 Thorsten Brach. All rights reserved                                                                                                                                            
//             Licensed under the LGPL-3.0 license.
//                                                                           
//  Disclaimer:                                                                           
//    This project is provided without any guarantee and can be used for   
//    private and commercial purposes. Any use is at the user’s 
//    own risk and responsibility.
//
// -------------------------------------------------------------------------
TYPE ArmConfigParameter :
STRUCT
  /// Configuration of shoulder
  Shoulder : ArmConfigShoulder;
  /// Configuration of elbow
  Elbow    : ArmConfigElbow;
  /// Configuration of wrist
  Wrist    : ArmConfigWrist;
END_STRUCT
END_TYPE

// Library/Structures/Miscellaneous/AuxOffset
{attribute 'pack_mode' := '1'} 
// ------------------------------------------------------------------------- 
//  SRCI Robot Library                                                
// ------------------------------------------------------------------------- 
//                                                                           
//  Object:      AuxOffset                                       
//  Author:      Thorsten Brach                                                
//  Date:        2024-06-01
//
//  Description:                                              
//   
//                                                                           
//  Copyright: 
//    (C) 2024 Thorsten Brach. All rights reserved                                                                                                                                            
//             Licensed under the LGPL-3.0 license.
//                                                                           
//  Disclaimer:                                                                           
//    This project is provided without any guarantee and can be used for   
//    private and commercial purposes. Any use is at the user’s 
//    own risk and responsibility.
//
// -------------------------------------------------------------------------
TYPE AuxOffset :
STRUCT
  /// Offset in X-Direction
  X  : REAL;
  /// Offset in Y-direction
  Y  : REAL;
  /// Offset in Z-direction
  Z  : REAL;
  /// Offset in Rx-Direction
  Rx : REAL;
  /// Offset in Ry-direction
  Ry : REAL;
  /// Offset in Rz-direction
  Rz : REAL;
END_STRUCT
END_TYPE

// Library/Structures/Miscellaneous/CoordinateSystem
{attribute 'pack_mode' := '1'} 
// ------------------------------------------------------------------------- 
//  SRCI Robot Library                                                
// ------------------------------------------------------------------------- 
//                                                                           
//  Object:      CoordinateSystem                                       
//  Author:      Thorsten Brach                                                
//  Date:        2024-06-01
//
//  Description:                                              
//   
//                                                                           
//  Copyright: 
//    (C) 2024 Thorsten Brach. All rights reserved                                                                                                                                            
//             Licensed under the LGPL-3.0 license.
//                                                                           
//  Disclaimer:                                                                           
//    This project is provided without any guarantee and can be used for   
//    private and commercial purposes. Any use is at the user’s 
//    own risk and responsibility.
//
// -------------------------------------------------------------------------
TYPE CoordinateSystem :
STRUCT
  /// Tool index
  /// • 0: Flange
  /// • 1..254: Tool frames
  ToolNo  : USINT;
  /// Frame index
  /// • 0: WCS
  /// • 1..254: User frames
  FrameNo : USINT;
END_STRUCT
END_TYPE

// Library/Structures/Miscellaneous/DataEnableSync
TYPE DataEnableSync :
{attribute 'pack_mode' := '1'} 
// ------------------------------------------------------------------------- 
//  SRCI Robot Library                                                
// ------------------------------------------------------------------------- 
//                                                                           
//  Object:      DataEnableSync                                       
//  Author:      Thorsten Brach                                                
//  Date:        2024-06-22
//
//  Description:                                              
//   
//                                                                           
//  Copyright: 
//    (C) 2024 Thorsten Brach. All rights reserved                                                                                                                                            
//             Licensed under the LGPL-3.0 license.
//                                                                           
//  Disclaimer:                                                                           
//    This project is provided without any guarantee and can be used for   
//    private and commercial purposes. Any use is at the user’s 
//    own risk and responsibility.
//
// -------------------------------------------------------------------------  
STRUCT
  /// Set TRUE (default), to activate the synchronizationrelated comparison mechanism for tool data
  EnableSyncTool              : BOOL;
  /// Set TRUE (default), to activate the synchronizationrelated comparison mechanism for frame data
  EnableSyncFrame             : BOOL;
  ///  Set TRUE (default), to activate the synchronizationrelated comparison mechanism for load data
  EnableSyncLoad              : BOOL;
  /// Set TRUE (default), to activate the synchronizationrelated comparison mechanism for work area data
  EnableSyncWorkArea          : BOOL;
  /// Set TRUE (default), to activate the synchronizationrelated comparison mechanism for software limits
  EnableSyncSWLimits          : BOOL;
  /// Set TRUE (default), to activate the synchronizationrelated comparison mechanism for default dynamics
  EnableSyncDefaultDynamics   : BOOL;
  /// Set TRUE (default), to activate the synchronizationrelated comparison mechanism for reference dynamics
  EnableSyncReferenceDynamics : BOOL;
  /// - Allows blending when CallSubprogram is called in sequence and removed afterwards.
  /// For more information see chapter 6.5.21.
  /// • 0 (default): Dynamic blending is prevented 
  /// • 1: Dynamic blending is allowed
  AllowDynamicBlending        : BOOL ;
END_STRUCT
END_TYPE

// Library/Structures/Miscellaneous/DataInSync
{attribute 'pack_mode' := '1'} 
// ------------------------------------------------------------------------- 
//  SRCI Robot Library                                                
// ------------------------------------------------------------------------- 
//                                                                           
//  Object:      DataInSync                                       
//  Author:      Thorsten Brach                                                
//  Date:        2024-06-01
//
//  Description:                                              
//   
//                                                                           
//  Copyright: 
//    (C) 2024 Thorsten Brach. All rights reserved                                                                                                                                            
//             Licensed under the LGPL-3.0 license.
//                                                                           
//  Disclaimer:                                                                           
//    This project is provided without any guarantee and can be used for   
//    private and commercial purposes. Any use is at the user’s 
//    own risk and responsibility.
//
// -------------------------------------------------------------------------
TYPE DataInSync :
STRUCT
  /// TRUE, if no tool has been modified
  ToolsInSync             : BOOL;
  /// TRUE, if no frame has been modified
  FramesInSync            : BOOL;
  /// TRUE, if no load has been modified
  LoadsInSync             : BOOL;
  /// TRUE, if no work area has been modified
  WorkAreasInSync         : BOOL;
  /// TRUE, if no software limit has been modified
  SoftwareLimitsInSync    : BOOL;
  /// TRUE, if no default dynamic parameter has been modified
  DefaultDynamicsInSync   : BOOL;
  /// TRUE, if no reference dynamic parameter has been modified
  ReferenceDynamicsInSync : BOOL;  
END_STRUCT
END_TYPE

// Library/Structures/Miscellaneous/DHParameter
{attribute 'pack_mode' := '1'} 
// ------------------------------------------------------------------------- 
//  SRCI Robot Library                                                
// ------------------------------------------------------------------------- 
//                                                                           
//  Object:      DHParameter                                       
//  Author:      Thorsten Brach                                                
//  Date:        2024-06-01
//
//  Description:                                              
//   
//                                                                           
//  Copyright: 
//    (C) 2024 Thorsten Brach. All rights reserved                                                                                                                                            
//             Licensed under the LGPL-3.0 license.
//                                                                           
//  Disclaimer:                                                                           
//    This project is provided without any guarantee and can be used for   
//    private and commercial purposes. Any use is at the user’s 
//    own risk and responsibility.
//
// -------------------------------------------------------------------------
TYPE DHParameter :
STRUCT
   /// DH parameter α for each joint - 0 If not supported
   Alpha                  : ARRAY [0..6] OF REAL;
   /// DH parameters A for each joint - 0 If not supported
   A                      : ARRAY [0..6] OF REAL;
   /// DH parameters D for each joint - 0 If not supported
   D                      : ARRAY [0..6] OF REAL;
   /// DH parameters Theta for each joint - 0 If not supported
   Theta                  : ARRAY [0..6] OF REAL;
   /// Positive joint direction of each joint. TRUE when positive joint direction points to the right.
   /// See also Figure 6-16.
   PositiveJointDirection : ARRAY [0..6] OF BOOL;
   /// Offset of zero position of joint to zero position suggested by Figure 6-17.
   JointZeroPosition      : ARRAY [0..6] OF REAL;
END_STRUCT
END_TYPE

// Library/Structures/Miscellaneous/ExternalAxesFlags
{attribute 'pack_mode' := '1'} 
// ------------------------------------------------------------------------- 
//  SRCI Robot Library                                                
// ------------------------------------------------------------------------- 
//                                                                           
//  Object:      ExternalAxesFlags                                       
//  Author:      Thorsten Brach                                                
//  Date:        2024-06-01
//
//  Description:                                              
//   
//                                                                           
//  Copyright: 
//    (C) 2024 Thorsten Brach. All rights reserved                                                                                                                                            
//             Licensed under the LGPL-3.0 license.
//                                                                           
//  Disclaimer:                                                                           
//    This project is provided without any guarantee and can be used for   
//    private and commercial purposes. Any use is at the user’s 
//    own risk and responsibility.
//
// -------------------------------------------------------------------------
TYPE ExternalAxesFlags :
STRUCT
  /// Bit 00 : Not used
  Bit00   : BOOL;
  /// Bit 01 : External axis E1 - property depends of usage 
  AxisE1  : BOOL;
  /// Bit 02 : External axis E2 - property depends of usage 
  AxisE2  : BOOL;
  /// Bit 03 : External axis E3 - property depends of usage 
  AxisE3  : BOOL;
  /// Bit 04 : External axis E4 - property depends of usage 
  AxisE4  : BOOL;
  /// Bit 05 : External axis E5 - property depends of usage 
  AxisE5  : BOOL;
  /// Bit 06 : External axis E6 - property depends of usage 
  AxisE6  : BOOL;
  /// Bit 00 : Not used
  Bit07   : BOOL;
END_STRUCT
END_TYPE

// Library/Structures/Miscellaneous/ForceStatus
{attribute 'pack_mode' := '1'} 
// ------------------------------------------------------------------------- 
//  SRCI Robot Library                                                
// ------------------------------------------------------------------------- 
//                                                                           
//  Object:      ForceStatus                                       
//  Author:      Thorsten Brach                                                
//  Date:        2024-06-01
//
//  Description:                                              
//   
//                                                                           
//  Copyright: 
//    (C) 2024 Thorsten Brach. All rights reserved                                                                                                                                            
//             Licensed under the LGPL-3.0 license.
//                                                                           
//  Disclaimer:                                                                           
//    This project is provided without any guarantee and can be used for   
//    private and commercial purposes. Any use is at the user’s 
//    own risk and responsibility.
//
// -------------------------------------------------------------------------
TYPE ForceStatus :
STRUCT
  /// TRUE, while a "ForceControl" function is enabled
  ForceControlEnabled         : BOOL;
  /// TRUE, while a "ForceLimit" function is enabled
  ForceLimitEnabled           : BOOL;
  /// TRUE, while robot is adjusting its movement to apply specified force
  ApplyingForce               : BOOL;
  /// TRUE, while maximum deviation according to input parameter "MaxDeviation" is reached
  MaxDeviationReached         : BOOL;
  /// TRUE, while currently applied force/torque is identical to specified force/torque
  SpecifiedForceTorqueReached : BOOL;
  /// TRUE, while currently detected force is identical to specified force limit
  SpecifiedForceLimitReached  : BOOL;
  /// Bit 06 Reserve
  Bit06                       : BOOL;
  /// Bit 07 Reserve
  Bit07                       : BOOL;  
END_STRUCT
END_TYPE

// Library/Structures/Miscellaneous/FragmentAction
{attribute 'pack_mode' := '1'} 
// ------------------------------------------------------------------------- 
//  SRCI Robot Library                                                
// ------------------------------------------------------------------------- 
//                                                                           
//  Object:      FragmentAction                                       
//  Author:      Thorsten Brach                                                
//  Date:        2024-06-01
//
//  Description:                                              
//   
//                                                                           
//  Copyright: 
//    (C) 2024 Thorsten Brach. All rights reserved                                                                                                                                            
//             Licensed under the LGPL-3.0 license.
//                                                                           
//  Disclaimer:                                                                           
//    This project is provided without any guarantee and can be used for   
//    private and commercial purposes. Any use is at the user’s 
//    own risk and responsibility.
//
// -------------------------------------------------------------------------
TYPE FragmentAction :
STRUCT
  /// Bit 00 : Command Message is completely received – Flag to trigger processing of the payload
  Complete : BOOL;
  /// Bit 01 :(only client->server): The first message fragment of a new CMD resets (set all ACR values of this CMD ID to 0) the ACR entry
  Reset    : BOOL;
  /// Bit 02: Clears the receiving buffer by setting all of its Bytes to 0.
  Clear    : BOOL;
  /// Bit 03
  BIT03    : BOOL;
  /// Bit 04
  BIT04    : BOOL;
  /// Bit 05
  BIT05    : BOOL;
  /// Bit 06
  BIT06    : BOOL;
  /// Bit 07
  BIT07    : BOOL;  
END_STRUCT
END_TYPE

// Library/Structures/Miscellaneous/JogControl
{attribute 'pack_mode' := '1'} 
// ------------------------------------------------------------------------- 
//  SRCI Robot Library                                                
// ------------------------------------------------------------------------- 
//                                                                           
//  Object:      JogControl                                       
//  Author:      Thorsten Brach                                                
//  Date:        2024-06-01
//
//  Description:                                              
//   
//                                                                           
//  Copyright: 
//    (C) 2024 Thorsten Brach. All rights reserved                                                                                                                                            
//             Licensed under the LGPL-3.0 license.
//                                                                           
//  Disclaimer:                                                                           
//    This project is provided without any guarantee and can be used for   
//    private and commercial purposes. Any use is at the user’s 
//    own risk and responsibility.
//
// -------------------------------------------------------------------------
TYPE JogControl :
STRUCT
  /// Mode Frame : Movement in positive direction X of selected frame
  /// Mode Tool  : Movement in positive direction X of selected tool
  /// Mode Axes  : Movement in positive direction joint 1
  X_J1_Pos  : BOOL;
  /// Mode Frame : Movement in negative direction X of selected frame
  /// Mode Tool  : Movement in negative direction X of selected tool
  /// Mode Axes  : Movement in negative direction joint 1
  X_J1_Neg  : BOOL;
  /// Mode Frame : Movement in positive direction Y of selected frame
  /// Mode Tool  : Movement in positive direction Y of selected tool
  /// Mode Axes  : Movement in positive direction joint 2
  Y_J2_Pos  : BOOL;
  /// Mode Frame : Movement in negative direction Y of selected frame
  /// Mode Tool  : Movement in negative direction Y of selected tool
  /// Mode Axes  : Movement in negative direction joint 2
  Y_J2_Neg  : BOOL;
  /// Mode Frame : Movement in positive direction Z of selected frame
  /// Mode Tool  : Movement in positive direction Z of selected tool
  /// Mode Axes  : Movement in positive direction joint 3
  Z_J3_Pos  : BOOL;
  /// Mode Frame : Movement in negative direction Z of selected frame
  /// Mode Tool  : Movement in negative direction Z of selected tool
  /// Mode Axes  : Movement in negative direction joint 3
  Z_J3_Neg  : BOOL;
  /// Mode Frame : Movement in positive direction Rx of selected frame
  /// Mode Tool  : Movement in positive direction Rx of selected tool
  /// Mode Axes  : Movement in positive direction joint 4
  Rx_J4_Pos : BOOL;
  /// Mode Frame : Movement in negative direction Rx of selected frame
  /// Mode Tool  : Movement in negative direction Rx of selected tool
  /// Mode Axes  : Movement in negative direction joint 4
  Rx_J4_Neg : BOOL;
  /// Mode Frame : Movement in positive direction Ry of selected frame
  /// Mode Tool  : Movement in positive direction Ry of selected tool
  /// Mode Axes  : Movement in positive direction joint 5
  Ry_J5_Pos : BOOL;
  /// Mode Frame : Movement in negative direction Ry of selected frame
  /// Mode Tool  : Movement in negative direction Ry of selected tool
  /// Mode Axes  : Movement in negative direction joint 5
  Ry_J5_Neg : BOOL;
  /// Mode Frame : Movement in positive direction Rz of selected frame
  /// Mode Tool  : Movement in positive direction Rz of selected tool
  /// Mode Axes  : Movement in positive direction joint 6
  Rz_J6_Pos : BOOL;
  /// Mode Frame : Movement in negative direction Rz of selected frame
  /// Mode Tool  : Movement in negative direction Rz of selected tool
  /// Mode Axes  : Movement in negative direction joint 6
  Rz_J6_Neg : BOOL;
  /// Mode Frame : not supported
  /// Mode Tool  : not supported
  /// Mode Axes  : Movement in positive direction first external axis
  E1_Pos    : BOOL;
  /// Mode Frame : not supported
  /// Mode Tool  : not supported
  /// Mode Axes  : Movement in negative direction first external axis
  E1_Neg    : BOOL;
  /// Mode Frame : not supported
  /// Mode Tool  : not supported
  /// Mode Axes  : Movement in positive direction second external axis
  E2_Pos    : BOOL;
  /// Mode Frame : not supported
  /// Mode Tool  : not supported
  /// Mode Axes  : Movement in negative direction second external axis
  E2_Neg    : BOOL;
  /// Mode Frame : not supported
  /// Mode Tool  : not supported
  /// Mode Axes  : Movement in positive direction third external axis
  E3_Pos    : BOOL;
  /// Mode Frame : not supported
  /// Mode Tool  : not supported
  /// Mode Axes  : Movement in negative direction third external axis
  E3_Neg    : BOOL;
  /// Mode Frame : not supported
  /// Mode Tool  : not supported
  /// Mode Axes  : Movement in positive direction fourth external axis
  E4_Pos    : BOOL;
  /// Mode Frame : not supported
  /// Mode Tool  : not supported
  /// Mode Axes  : Movement in negative direction fourth external axis
  E4_Neg    : BOOL;
  /// Mode Frame : not supported
  /// Mode Tool  : not supported
  /// Mode Axes  : Movement in positive direction fifth external axis
  E5_Pos    : BOOL;
  /// Mode Frame : not supported
  /// Mode Tool  : not supported
  /// Mode Axes  : Movement in negative direction fifth external axis
  E5_Neg    : BOOL;
  /// Mode Frame : not supported
  /// Mode Tool  : not supported
  /// Mode Axes  : Movement in positive direction sixth external axis
  E6_Pos    : BOOL;
  /// Mode Frame : not supported
  /// Mode Tool  : not supported
  /// Mode Axes  : Movement in negative direction sixts external axis
  E6_Neg    : BOOL;
  
END_STRUCT
END_TYPE

// Library/Structures/Miscellaneous/MeasuringInputResult
{attribute 'pack_mode' := '1'} 
// ------------------------------------------------------------------------- 
//  SRCI Robot Library                                                
// ------------------------------------------------------------------------- 
//                                                                           
//  Object:      MeasuringInputResult                                       
//  Author:      Thorsten Brach                                                
//  Date:        2024-06-01
//
//  Description:                                              
//   
//                                                                           
//  Copyright: 
//    (C) 2024 Thorsten Brach. All rights reserved                                                                                                                                            
//             Licensed under the LGPL-3.0 license.
//                                                                           
//  Disclaimer:                                                                           
//    This project is provided without any guarantee and can be used for   
//    private and commercial purposes. Any use is at the user’s 
//    own risk and responsibility.
//
// -------------------------------------------------------------------------
TYPE MeasuringInputResult :
STRUCT
  /// Measured robot position value at the rising edge of the digital input in selected coordinate systems (see input parameters ToolNo and FrameNo).
  MeasuredCartesianPosition :  RobotCartesianPosition;
  /// Index of tool of returned position
  /// • 0: Flange
  /// • 1..254: Tool frames
  ToolNo                    : USINT;
  /// Index of frame of returned position
  /// • 0: WCS
  /// • 1..254: User frames
  FrameNo                   : USINT;
  /// Measured robot position value at the rising edge of the digital input in Joint position.
  MeasuredJointPosition     : RobotJointPosition;
END_STRUCT
END_TYPE

// Library/Structures/Miscellaneous/ProcessingModeAllowed
{attribute 'pack_mode' := '1'} 
// ------------------------------------------------------------------------- 
//  SRCI Robot Library                                                
// ------------------------------------------------------------------------- 
//                                                                           
//  Object:      ProcessingModeAllowed                                       
//  Author:      Thorsten Brach                                                
//  Date:        2024-06-01
//
//  Description:                                              
//   
//                                                                           
//  Copyright: 
//    (C) 2024 Thorsten Brach. All rights reserved                                                                                                                                            
//             Licensed under the LGPL-3.0 license.
//                                                                           
//  Disclaimer:                                                                           
//    This project is provided without any guarantee and can be used for   
//    private and commercial purposes. Any use is at the user’s 
//    own risk and responsibility.
//
// -------------------------------------------------------------------------
TYPE ProcessingModeAllowed :
STRUCT
  /// Command is buffered in sequence buffer and executed once
  BUFFERED           : BOOL;
  /// Command is buffered in sequence buffer, aborts and empties previous commands in sequence buffer, and is executed once
  ABORTING           : BOOL;
  /// Command is buffered in parallel buffer and executed once
  PARALLEL           : BOOL;
  /// Command is buffered in parallel buffer and executed repeatedly until deliberate deactivation by user
  CONTINUOUS         : BOOL;
  /// CMD execution is stopped and/or CMD is removed from the buffer
  DEACTIVATE         : BOOL;
  /// Command is buffered in sequence buffer and executed once (Trigger based)
  TRIGGER_BUFFERED   : BOOL;
  /// Command is buffered in sequence buffer, aborts and empties previous commands in sequence buffer, and is executed once (Trigger based)
  TRIGGER_ABORTING   : BOOL;
  /// Command is buffered in parallel buffer and executed once (Trigger based)
  TRIGGER_ONCE       : BOOL;
  /// Command is buffered in parallel buffer and executed repeatedly until deliberate deactivation by user (Trigger based)
  TRIGGER_CONTINUOUS : BOOL;
  /// Command is buffered and executed multiple times when triggered. The CMD remains in the buffer until removed by the user.
  TRIGGER_MULTIPLE   : BOOL;  
END_STRUCT
END_TYPE

// Library/Structures/Miscellaneous/RaStatusWord
{attribute 'pack_mode' := '1'} 
// ------------------------------------------------------------------------- 
//  SRCI Robot Library                                                
// ------------------------------------------------------------------------- 
//                                                                           
//  Object:      RaStatusWord                                       
//  Author:      Thorsten Brach                                                
//  Date:        2024-06-01
//
//  Description:                                              
//   
//                                                                           
//  Copyright: 
//    (C) 2024 Thorsten Brach. All rights reserved                                                                                                                                            
//             Licensed under the LGPL-3.0 license.
//                                                                           
//  Disclaimer:                                                                           
//    This project is provided without any guarantee and can be used for   
//    private and commercial purposes. Any use is at the user’s 
//    own risk and responsibility.
//
// -------------------------------------------------------------------------
TYPE RaStatusWord :
STRUCT
  /// Bit 00: 
  /// TRUE, when robot’s axes values change due to physical movement of axes
  IsMoving                 : BOOL;
  /// Bit 01: 
  /// TRUE, when move commands buffered by the primary sequence are currently not processed
  PrimarySequencePaused    : BOOL;
  /// Bit 02: 
  /// TRUE, when robot is moving in the primary sequence, FALSE when robot leaves its position by other means
  /// Switches back to TRUE in the following two scenarios:
  /// 1. During a change to the primary sequence the current TCP position is equal to
  ///    - position when the primary sequence was left
  ///    - target position of an interrupted move command of the primary sequence (see "ReturnToPrimary": "ReturnMode" "End position" chapter 6.3.11)
  /// 2. The primary sequence is active, and the buffer is empty while a new command is buffered by the primary sequence
  /// Independent of RA state
  InPrimaryPos             : BOOL;
  /// Bit 03:
  /// Secondary sequence is active, either by user selection or by implicit behavior
  SecondarySequenceActive  : BOOL;
  /// Bit 04:
  /// TRUE, when robot is currently blending between two move commands
  IsBlending               : BOOL;
  /// Bit 05:
  /// Shows that an error acknowledgement by the client is necessary
  ErrorPending             : BOOL;
  /// Bit 06:
  /// RC is restarting
  RestartInProgress        : BOOL;
  /// Bit 07:
  /// RA power state
  Enabled                  : BOOL;
  /// Bit 08 - 09: RA sequence states: Idle, Interrupt active, Axes controlled
  RaSequenceState          : RaSequenceState;
  /// Bit 10 - Bit 12:
  /// Operation Mode: T1 Local, T2 Local, Auto, Auto Ext, T1 Ext, T2 Ext
  OperationMode            : OperationMode;
  /// Bit 13:
  /// TRUE, while CollisionDetection is enabled (see chapter 6.5.35) 
  CollisionDetectedEnabled : BOOL;
  /// Bit 14:
  /// TRUE, when a collision was detected while CollisionDetection is enabled
  CollisionDetected        : BOOL;
  /// Bit 15:
  /// TRUE, when the RC request a restart of the RCinduced through the functions "WriteRobotSWLimits" or "WriteSystemVariable"
  RestartRequested         : BOOL;
  /// Bit 16:
  /// RA is currently accelerating. Support of this value is returned via exchangeConfig.
  Accelerating             : BOOL;
  /// Bit 17:
  /// RA is currently decelerating. Support of this value is returned via exchangeConfig.
  Decelerating             : BOOL;
  /// Bit 18:
  /// RA is currently not accelerating nor decelerating. Support of this value is returned via exchangeConfig.
  ConstantVelocity         : BOOL;
  /// Bit 19
  Bit19                    : BOOL;
  /// Bit 20
  Bit20                    : BOOL;
  /// Bit 21
  Bit21                    : BOOL;
  /// Bit 22
  Bit22                    : BOOL;
  /// Bit 23
  Bit23                    : BOOL;
  /// Bit 24
  Bit24                    : BOOL;
  /// Bit 25
  Bit25                    : BOOL;
  /// Bit 26
  Bit26                    : BOOL;
  /// Bit 27
  Bit27                    : BOOL;
  /// Bit 28
  Bit28                    : BOOL;
  /// Bit 29
  Bit29                    : BOOL;
  /// Bit 30
  Bit30                    : BOOL;
  /// Bit 31
  Bit31                    : BOOL;  
END_STRUCT
END_TYPE

